FUNCTION CheckDivWord : WORD
VAR_INPUT
	divisor				: WORD;
END_VAR
VAR
END_VAR

IF divisor = 0 THEN
	CheckWordZeroDiv_ErrCnt:= CheckWordZeroDiv_ErrCnt + 1;
	CheckDivWord := 1;
ELSE
	CheckDivWord := divisor;
END_IF

END_FUNCTION

(* stored: Version 1.1.0.1, ProductVersion 3.1.4024.9
   POU CheckDivWord: Id {496dbc3e-4bce-4ac7-97b2-5489846ca8c7}, SpecialFunc CheckDivInt32 *)
